// TIA Portal project "Styringsenhed" (V13)

(* hardware
DEVICE "S7-1200 station_1"  S7-1200 Station
   slot 0: "Rack_0"  Rack  V1.0
   slot 1: "PLC_1"  CPU 1214C DC/DC/DC  6ES7 214-1AG40-0XB0  V4.1
   slot 3: "AQ 1x12BIT_1"  6ES7 232-4HA30-0XB0  V1.0
DEVICE "HMI_1"  KTP600 Basic color PN
   slot 0: "HMI"  HMI  6AV6 647-0AD11-3AX0  12.0.0.0
   slot 1: "HMI_RT_1"  KTP600 Basic color PN  6AV6 647-0AD11-3AX0  12.0.0.0
   slot 5: "HMI_1.IE_CP_1"  PROFINET Interface
      slot 1: "PROFINET Interface_1"  PROFINET Interface
         slot 1: "Port_1"  Port
*)

// ===== PLC "PLC_1"  CPU 1214C DC/DC/DC =====

DATA_BLOCK "EthernetDB"   // DB3
{ S7_Optimized_Access := 'FALSE' }
VERSION : 0.1
   VAR
      "Start_request(REQ)" : Bool;
      "Connection_state(CONT)" : Bool;
      "Send_length(LEN)" : UInt;
      "Send_area(DATA)" : String;
      "Restart_block(COM_RST)" : Bool;
      "Request_completion(DONE)" : Bool;
      "Request_processing(BUSY)" : Bool;
      "Error(ERROR)" : Bool;
      "Error_information(STATUS)" : Word;
   END_VAR
BEGIN
END_DATA_BLOCK

// folder: System blocks/Program resources

DATA_BLOCK "PLC_1_Send_DB"   // DB2
{ S7_Optimized_Access := 'FALSE' }
AUTHOR : SIMATIC
FAMILY : MC7Plus
NAME : TC_IP_v4
VERSION : 1.0
// stored: InstanceOfName ?
"?"
BEGIN
END_DATA_BLOCK

// folder: (top level)

FUNCTION "Ethernet" : Void   // FC1, LAD
{ S7_Optimized_Access := 'FALSE' }
VERSION : 0.1
BEGIN

REGION Network 1
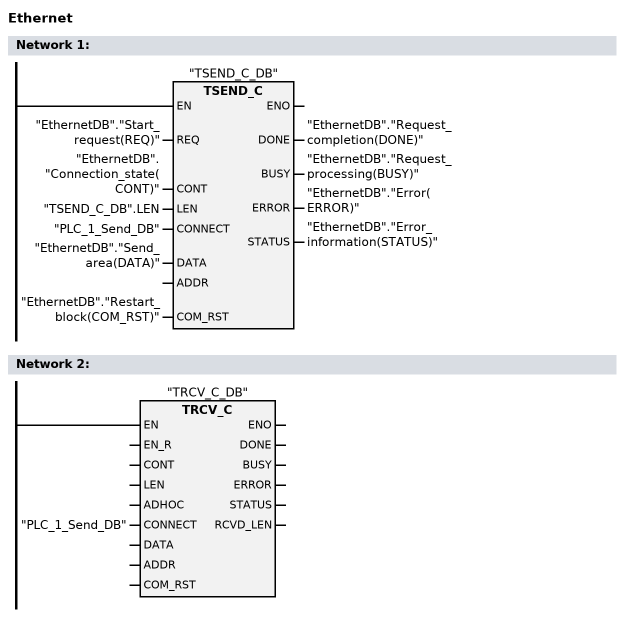
   "TSEND_C_DB"(REQ := "EthernetDB"."Start_request(REQ)",   // TSEND_C
                CONT := "EthernetDB"."Connection_state(CONT)",
                LEN := "TSEND_C_DB".LEN,
                CONNECT := "PLC_1_Send_DB",
                DATA := "EthernetDB"."Send_area(DATA)",
                COM_RST := "EthernetDB"."Restart_block(COM_RST)",
                DONE => "EthernetDB"."Request_completion(DONE)",
                BUSY => "EthernetDB"."Request_processing(BUSY)",
                ERROR => "EthernetDB"."Error(ERROR)",
                STATUS => "EthernetDB"."Error_information(STATUS)");
END_REGION

REGION Network 2
   "TRCV_C_DB"(CONNECT := "PLC_1_Send_DB");   // TRCV_C
END_REGION
END_FUNCTION

ORGANIZATION_BLOCK "Main"   // OB1, LAD, ProgramCycle
TITLE = "Main Program Sweep (Cycle)"
{ S7_Optimized_Access := 'FALSE' }
VERSION : 0.1
BEGIN
END_ORGANIZATION_BLOCK